ABB RAPID module: Module1.mod

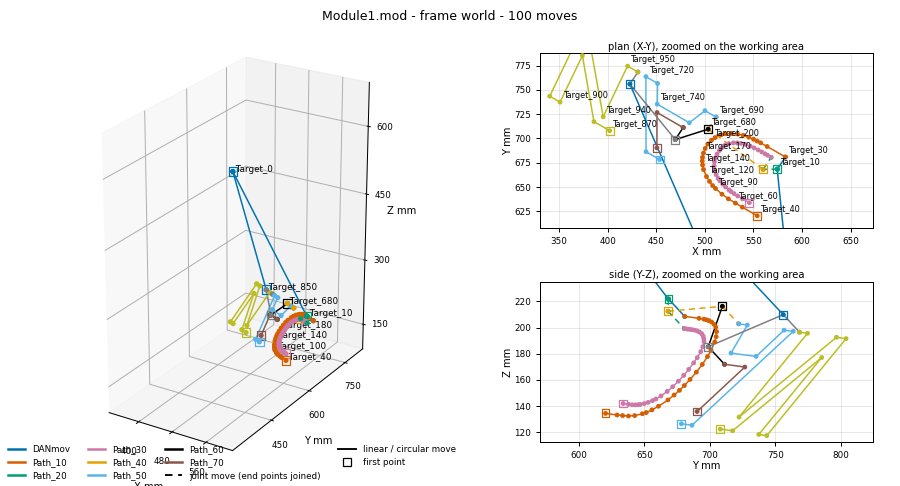
[picture p0: tool path of Module1.mod in frame world, 100 of 100 moves have a stored position in this frame; points joined in program order, loops and branches not executed]
MODULE Module1
        CONST robtarget Target_20:=[[0.071,0.06,-20],[1,0,0,0],[0,0,0,0],[9E+09,9E+09,9E+09,9E+09,9E+09,9E+09]];
    CONST robtarget Target_30:=[[0.095,0.07,0],[1,0,0,0],[0,0,0,0],[9E+09,9E+09,9E+09,9E+09,9E+09,9E+09]];
    CONST robtarget Target_40:=[[99.94,0.237,0],[1,0,0,0],[0,0,0,0],[9E+09,9E+09,9E+09,9E+09,9E+09,9E+09]];
    CONST robtarget Target_50:=[[99.89,17.95,0],[1,0,0,0],[0,0,0,0],[9E+09,9E+09,9E+09,9E+09,9E+09,9E+09]];
    CONST robtarget Target_60:=[[99.72,26.211,0],[1,0,0,0],[0,0,0,0],[9E+09,9E+09,9E+09,9E+09,9E+09,9E+09]];
    CONST robtarget Target_70:=[[99.369,34.775,0],[1,0,0,0],[0,0,0,0],[9E+09,9E+09,9E+09,9E+09,9E+09,9E+09]];
    CONST robtarget Target_80:=[[98.151,42.817,0],[1,0,0,0],[0,0,0,0],[9E+09,9E+09,9E+09,9E+09,9E+09,9E+09]];
    CONST robtarget Target_90:=[[95.465,51.41,0],[1,0,0,0],[0,0,0,0],[9E+09,9E+09,9E+09,9E+09,9E+09,9E+09]];
    CONST robtarget Target_100:=[[93.827,55.395,0],[1,0,0,0],[0,0,0,0],[9E+09,9E+09,9E+09,9E+09,9E+09,9E+09]];
    CONST robtarget Target_110:=[[90.626,60.139,0],[1,0,0,0],[0,0,0,0],[9E+09,9E+09,9E+09,9E+09,9E+09,9E+09]];
    CONST robtarget Target_120:=[[86.457,65.135,0],[1,0,0,0],[0,0,0,0],[9E+09,9E+09,9E+09,9E+09,9E+09,9E+09]];
    CONST robtarget Target_130:=[[79.404,71.019,0],[1,0,0,0],[0,0,0,0],[9E+09,9E+09,9E+09,9E+09,9E+09,9E+09]];
    CONST robtarget Target_140:=[[74.069,73.954,0],[1,0,0,0],[0,0,0,0],[9E+09,9E+09,9E+09,9E+09,9E+09,9E+09]];
    CONST robtarget Target_150:=[[69.003,75.99,0],[1,0,0,0],[0,0,0,0],[9E+09,9E+09,9E+09,9E+09,9E+09,9E+09]];
    CONST robtarget Target_160:=[[63.952,77.379,0],[1,0,0,0],[0,0,0,0],[9E+09,9E+09,9E+09,9E+09,9E+09,9E+09]];
    CONST robtarget Target_170:=[[57.546,78.369,0],[1,0,0,0],[0,0,0,0],[9E+09,9E+09,9E+09,9E+09,9E+09,9E+09]];
    CONST robtarget Target_180:=[[50.002,78.831,0],[1,0,0,0],[0,0,0,0],[9E+09,9E+09,9E+09,9E+09,9E+09,9E+09]];
    CONST robtarget Target_190:=[[42.114,78.338,0],[1,0,0,0],[0,0,0,0],[9E+09,9E+09,9E+09,9E+09,9E+09,9E+09]];
    CONST robtarget Target_200:=[[34.188,76.601,0],[1,0,0,0],[0,0,0,0],[9E+09,9E+09,9E+09,9E+09,9E+09,9E+09]];
    CONST robtarget Target_210:=[[27.953,74.421,0],[1,0,0,0],[0,0,0,0],[9E+09,9E+09,9E+09,9E+09,9E+09,9E+09]];
    CONST robtarget Target_220:=[[19.688,70.032,0],[1,0,0,0],[0,0,0,0],[9E+09,9E+09,9E+09,9E+09,9E+09,9E+09]];
    CONST robtarget Target_230:=[[14.672,66.13,0],[1,0,0,0],[0,0,0,0],[9E+09,9E+09,9E+09,9E+09,9E+09,9E+09]];
    CONST robtarget Target_240:=[[9.923,60.959,0],[1,0,0,0],[0,0,0,0],[9E+09,9E+09,9E+09,9E+09,9E+09,9E+09]];
    CONST robtarget Target_250:=[[5.883,54.79,0],[1,0,0,0],[0,0,0,0],[9E+09,9E+09,9E+09,9E+09,9E+09,9E+09]];
    CONST robtarget Target_260:=[[3.458,49.141,0],[1,0,0,0],[0,0,0,0],[9E+09,9E+09,9E+09,9E+09,9E+09,9E+09]];
    CONST robtarget Target_270:=[[1.636,43.084,0],[1,0,0,0],[0,0,0,0],[9E+09,9E+09,9E+09,9E+09,9E+09,9E+09]];
    CONST robtarget Target_280:=[[0.741,37.699,0],[1,0,0,0],[0,0,0,0],[9E+09,9E+09,9E+09,9E+09,9E+09,9E+09]];
    CONST robtarget Target_290:=[[0.334,33.582,0],[1,0,0,0],[0,0,0,0],[9E+09,9E+09,9E+09,9E+09,9E+09,9E+09]];
    CONST robtarget Target_300:=[[0.083,29.539,0],[1,0,0,0],[0,0,0,0],[9E+09,9E+09,9E+09,9E+09,9E+09,9E+09]];
    CONST robtarget Target_310:=[[-0.058,21.739,0],[1,0,0,0],[0,0,0,0],[9E+09,9E+09,9E+09,9E+09,9E+09,9E+09]];
    CONST robtarget Target_320:=[[-0.012,0.002,0],[1,0,0,0],[0,0,0,0],[9E+09,9E+09,9E+09,9E+09,9E+09,9E+09]];
    CONST robtarget Target_330:=[[0.01,0.019,-20],[1,0,0,0],[0,0,0,0],[9E+09,9E+09,9E+09,9E+09,9E+09,9E+09]];
    CONST robtarget Target_340:=[[11.428,13.269,-20],[1,0,0,0],[0,0,0,0],[9E+09,9E+09,9E+09,9E+09,9E+09,9E+09]];
    CONST robtarget Target_350:=[[11.415,13.206,0],[1,0,0,0],[0,0,0,0],[9E+09,9E+09,9E+09,9E+09,9E+09,9E+09]];
    CONST robtarget Target_360:=[[88.506,13.381,0],[1,0,0,0],[0,0,0,0],[9E+09,9E+09,9E+09,9E+09,9E+09,9E+09]];
    CONST robtarget Target_370:=[[88.487,21.649,0],[1,0,0,0],[0,0,0,0],[9E+09,9E+09,9E+09,9E+09,9E+09,9E+09]];
    CONST robtarget Target_380:=[[88.485,27.345,0],[1,0,0,0],[0,0,0,0],[9E+09,9E+09,9E+09,9E+09,9E+09,9E+09]];
    CONST robtarget Target_390:=[[88.109,31.752,0],[1,0,0,0],[0,0,0,0],[9E+09,9E+09,9E+09,9E+09,9E+09,9E+09]];
    CONST robtarget Target_400:=[[87.669,35.444,0],[1,0,0,0],[0,0,0,0],[9E+09,9E+09,9E+09,9E+09,9E+09,9E+09]];
    CONST robtarget Target_410:=[[87.109,38.017,0],[1,0,0,0],[0,0,0,0],[9E+09,9E+09,9E+09,9E+09,9E+09,9E+09]];
    CONST robtarget Target_420:=[[85.774,42.593,0],[1,0,0,0],[0,0,0,0],[9E+09,9E+09,9E+09,9E+09,9E+09,9E+09]];
    CONST robtarget Target_430:=[[84.168,46.535,0],[1,0,0,0],[0,0,0,0],[9E+09,9E+09,9E+09,9E+09,9E+09,9E+09]];
    CONST robtarget Target_440:=[[81.999,50.598,0],[1,0,0,0],[0,0,0,0],[9E+09,9E+09,9E+09,9E+09,9E+09,9E+09]];
    CONST robtarget Target_450:=[[80.078,53.34,0],[1,0,0,0],[0,0,0,0],[9E+09,9E+09,9E+09,9E+09,9E+09,9E+09]];
    CONST robtarget Target_460:=[[76.624,56.897,0],[1,0,0,0],[0,0,0,0],[9E+09,9E+09,9E+09,9E+09,9E+09,9E+09]];
    CONST robtarget Target_470:=[[71.616,60.336,0],[1,0,0,0],[0,0,0,0],[9E+09,9E+09,9E+09,9E+09,9E+09,9E+09]];
    CONST robtarget Target_480:=[[66.489,62.685,0],[1,0,0,0],[0,0,0,0],[9E+09,9E+09,9E+09,9E+09,9E+09,9E+09]];
    CONST robtarget Target_490:=[[60.688,64.314,0],[1,0,0,0],[0,0,0,0],[9E+09,9E+09,9E+09,9E+09,9E+09,9E+09]];
    CONST robtarget Target_500:=[[54.646,65.083,0],[1,0,0,0],[0,0,0,0],[9E+09,9E+09,9E+09,9E+09,9E+09,9E+09]];
    CONST robtarget Target_510:=[[48.445,65.222,0],[1,0,0,0],[0,0,0,0],[9E+09,9E+09,9E+09,9E+09,9E+09,9E+09]];
    CONST robtarget Target_520:=[[41.793,64.617,0],[1,0,0,0],[0,0,0,0],[9E+09,9E+09,9E+09,9E+09,9E+09,9E+09]];
    CONST robtarget Target_530:=[[36.504,63.714,0],[1,0,0,0],[0,0,0,0],[9E+09,9E+09,9E+09,9E+09,9E+09,9E+09]];
    CONST robtarget Target_540:=[[30.458,61.691,0],[1,0,0,0],[0,0,0,0],[9E+09,9E+09,9E+09,9E+09,9E+09,9E+09]];
    CONST robtarget Target_550:=[[25.646,58.958,0],[1,0,0,0],[0,0,0,0],[9E+09,9E+09,9E+09,9E+09,9E+09,9E+09]];
    CONST robtarget Target_560:=[[20.836,54.923,0],[1,0,0,0],[0,0,0,0],[9E+09,9E+09,9E+09,9E+09,9E+09,9E+09]];
    CONST robtarget Target_570:=[[18.13,51.34,0],[1,0,0,0],[0,0,0,0],[9E+09,9E+09,9E+09,9E+09,9E+09,9E+09]];
    CONST robtarget Target_580:=[[15.883,47.659,0],[1,0,0,0],[0,0,0,0],[9E+09,9E+09,9E+09,9E+09,9E+09,9E+09]];
    CONST robtarget Target_590:=[[13.855,43.017,0],[1,0,0,0],[0,0,0,0],[9E+09,9E+09,9E+09,9E+09,9E+09,9E+09]];
    CONST robtarget Target_600:=[[12.476,37.696,0],[1,0,0,0],[0,0,0,0],[9E+09,9E+09,9E+09,9E+09,9E+09,9E+09]];
    CONST robtarget Target_610:=[[11.809,33.29,0],[1,0,0,0],[0,0,0,0],[9E+09,9E+09,9E+09,9E+09,9E+09,9E+09]];
    CONST robtarget Target_620:=[[11.395,28.602,0],[1,0,0,0],[0,0,0,0],[9E+09,9E+09,9E+09,9E+09,9E+09,9E+09]];
    CONST robtarget Target_630:=[[11.309,24.432,0],[1,0,0,0],[0,0,0,0],[9E+09,9E+09,9E+09,9E+09,9E+09,9E+09]];
    CONST robtarget Target_640:=[[11.306,20.553,0],[1,0,0,0],[0,0,0,0],[9E+09,9E+09,9E+09,9E+09,9E+09,9E+09]];
    CONST robtarget Target_650:=[[11.368,17.578,0],[1,0,0,0],[0,0,0,0],[9E+09,9E+09,9E+09,9E+09,9E+09,9E+09]];
    CONST robtarget Target_660:=[[11.3,13.377,0],[1,0,0,0],[0,0,0,0],[9E+09,9E+09,9E+09,9E+09,9E+09,9E+09]];
    CONST robtarget Target_670:=[[11.431,13.345,-20],[1,0,0,0],[0,0,0,0],[9E+09,9E+09,9E+09,9E+09,9E+09,9E+09]];
    CONST robtarget Target_680:=[[-0.137,82.54,-20],[1,0,0,0],[0,0,0,0],[9E+09,9E+09,9E+09,9E+09,9E+09,9E+09]];
    CONST robtarget Target_690:=[[-0.154,82.529,0],[1,0,0,0],[0,0,0,0],[9E+09,9E+09,9E+09,9E+09,9E+09,9E+09]];
    CONST robtarget Target_700:=[[99.658,116.481,0],[1,0,0,0],[0,0,0,0],[9E+09,9E+09,9E+09,9E+09,9E+09,9E+09]];
    CONST robtarget Target_710:=[[99.61,132.697,0],[1,0,0,0],[0,0,0,0],[9E+09,9E+09,9E+09,9E+09,9E+09,9E+09]];
    CONST robtarget Target_720:=[[-0.345,166.23,0],[1,0,0,0],[0,0,0,0],[9E+09,9E+09,9E+09,9E+09,9E+09,9E+09]];
    CONST robtarget Target_730:=[[-0.179,152.289,0],[1,0,0,0],[0,0,0,0],[9E+09,9E+09,9E+09,9E+09,9E+09,9E+09]];
    CONST robtarget Target_740:=[[27.683,143.366,0],[1,0,0,0],[0,0,0,0],[9E+09,9E+09,9E+09,9E+09,9E+09,9E+09]];
    CONST robtarget Target_750:=[[27.893,105.098,0],[1,0,0,0],[0,0,0,0],[9E+09,9E+09,9E+09,9E+09,9E+09,9E+09]];
    CONST robtarget Target_760:=[[-0.159,95.872,0],[1,0,0,0],[0,0,0,0],[9E+09,9E+09,9E+09,9E+09,9E+09,9E+09]];
    CONST robtarget Target_770:=[[-0.14,82.55,0],[1,0,0,0],[0,0,0,0],[9E+09,9E+09,9E+09,9E+09,9E+09,9E+09]];
    CONST robtarget Target_780:=[[-0.154,82.561,-20],[1,0,0,0],[0,0,0,0],[9E+09,9E+09,9E+09,9E+09,9E+09,9E+09]];
    CONST robtarget Target_790:=[[39.082,108.722,-20],[1,0,0,0],[0,0,0,0],[9E+09,9E+09,9E+09,9E+09,9E+09,9E+09]];
    CONST robtarget Target_800:=[[39.077,108.691,0],[1,0,0,0],[0,0,0,0],[9E+09,9E+09,9E+09,9E+09,9E+09,9E+09]];
    CONST robtarget Target_810:=[[86.241,124.237,0],[1,0,0,0],[0,0,0,0],[9E+09,9E+09,9E+09,9E+09,9E+09,9E+09]];
    CONST robtarget Target_820:=[[38.992,139.852,0],[1,0,0,0],[0,0,0,0],[9E+09,9E+09,9E+09,9E+09,9E+09,9E+09]];
    CONST robtarget Target_830:=[[39.046,108.686,0],[1,0,0,0],[0,0,0,0],[9E+09,9E+09,9E+09,9E+09,9E+09,9E+09]];
    CONST robtarget Target_840:=[[39.049,108.56,-20],[1,0,0,0],[0,0,0,0],[9E+09,9E+09,9E+09,9E+09,9E+09,9E+09]];
    CONST robtarget Target_850:=[[-0.358,175.771,-20],[1,0,0,0],[0,0,0,0],[9E+09,9E+09,9E+09,9E+09,9E+09,9E+09]];
    CONST robtarget Target_860:=[[-0.349,175.774,0],[1,0,0,0],[0,0,0,0],[9E+09,9E+09,9E+09,9E+09,9E+09,9E+09]];
    CONST robtarget Target_870:=[[99.545,176.056,0],[1,0,0,0],[0,0,0,0],[9E+09,9E+09,9E+09,9E+09,9E+09,9E+09]];
    CONST robtarget Target_880:=[[99.462,194.82,0],[1,0,0,0],[0,0,0,0],[9E+09,9E+09,9E+09,9E+09,9E+09,9E+09]];
    CONST robtarget Target_890:=[[20.206,234.954,0],[1,0,0,0],[0,0,0,0],[9E+09,9E+09,9E+09,9E+09,9E+09,9E+09]];
    CONST robtarget Target_900:=[[99.467,235.15,0],[1,0,0,0],[0,0,0,0],[9E+09,9E+09,9E+09,9E+09,9E+09,9E+09]];
    CONST robtarget Target_910:=[[99.468,247.445,0],[1,0,0,0],[0,0,0,0],[9E+09,9E+09,9E+09,9E+09,9E+09,9E+09]];
    CONST robtarget Target_920:=[[-0.422,247.2,0],[1,0,0,0],[0,0,0,0],[9E+09,9E+09,9E+09,9E+09,9E+09,9E+09]];
    CONST robtarget Target_930:=[[-0.414,232.573,0],[1,0,0,0],[0,0,0,0],[9E+09,9E+09,9E+09,9E+09,9E+09,9E+09]];
    CONST robtarget Target_940:=[[85.947,188.296,0],[1,0,0,0],[0,0,0,0],[9E+09,9E+09,9E+09,9E+09,9E+09,9E+09]];
    CONST robtarget Target_950:=[[-0.342,188.055,0],[1,0,0,0],[0,0,0,0],[9E+09,9E+09,9E+09,9E+09,9E+09,9E+09]];
    CONST robtarget Target_960:=[[-0.342,175.796,0],[1,0,0,0],[0,0,0,0],[9E+09,9E+09,9E+09,9E+09,9E+09,9E+09]];
    CONST robtarget Target_970:=[[-0.334,175.799,-20],[1,0,0,0],[0,0,0,0],[9E+09,9E+09,9E+09,9E+09,9E+09,9E+09]];
    CONST robtarget Target_0:=[[-134.031,-231.216,-517.135],[1,0,0,0],[0,0,-1,0],[9E+09,9E+09,9E+09,9E+09,9E+09,9E+09]];
    CONST robtarget Target_10:=[[0.269,0.222,-20],[1,0,0,0],[0,0,0,0],[9E+09,9E+09,9E+09,9E+09,9E+09,9E+09]];
    CONST robtarget Target_1000:=[[-134.031,-231.216,-517.135],[1,0,0,0],[0,0,-1,0],[9E+09,9E+09,9E+09,9E+09,9E+09,9E+09]];
        TASK PERS wobjdata DANinclindo:=[FALSE,TRUE,"",[[0,0,10],[1,0,0,0]],[[366.1,610.764,198.883],[0.288677,-0.643742,0.654749,0.271228]]];
!***********************************************************
    !
    ! Módulo:  Module1
    !
    ! Descripción:
    !   <Introduzca la descripción aquí>
    !
    ! Autor: Danilo
    !
    ! Versión: 1.0
    !
    !***********************************************************


    !***********************************************************
    !
    ! Procedimiento Main
    !
    !   Este es el punto de entrada de su programa
    !
    !***********************************************************
    PROC main()
        !Añada aquí su código
        DANmov;
        Path_10;
        Path_20;
        Path_30;
        Path_40;
        Path_50;
        Path_60;
        Path_70;
        Path_80;
        Path_90;
        Path_100;
    ENDPROC
    PROC DANmov()
        MoveL Target_0,v100,z10,MARCADORBIEN\WObj:=DAN;
        MoveL Target_10,v100,z10,MARCADORBIEN\WObj:=DAN;
        MoveL Target_20,v100,z10,MARCADORBIEN\WObj:=DAN;
        MoveL Target_30,v100,z10,MARCADORBIEN\WObj:=DAN;
    ENDPROC
    PROC Path_10()
        MoveL Target_40,v100,z10,MARCADORBIEN\WObj:=DAN;
        MoveL Target_50,v100,z10,MARCADORBIEN\WObj:=DAN;
        MoveL Target_60,v100,z10,MARCADORBIEN\WObj:=DAN;
        MoveL Target_70,v100,z10,MARCADORBIEN\WObj:=DAN;
        MoveL Target_80,v100,z10,MARCADORBIEN\WObj:=DAN;
        MoveL Target_90,v100,z10,MARCADORBIEN\WObj:=DAN;
        MoveL Target_100,v100,z10,MARCADORBIEN\WObj:=DAN;
        MoveL Target_110,v100,z10,MARCADORBIEN\WObj:=DAN;
        MoveL Target_120,v100,z10,MARCADORBIEN\WObj:=DAN;
        MoveL Target_130,v100,z10,MARCADORBIEN\WObj:=DAN;
        MoveL Target_140,v100,z10,MARCADORBIEN\WObj:=DAN;
        MoveL Target_150,v100,z10,MARCADORBIEN\WObj:=DAN;
        MoveL Target_160,v100,z10,MARCADORBIEN\WObj:=DAN;
        MoveL Target_170,v100,z10,MARCADORBIEN\WObj:=DAN;
        MoveL Target_180,v100,z10,MARCADORBIEN\WObj:=DAN;
        MoveL Target_190,v100,z10,MARCADORBIEN\WObj:=DAN;
        MoveL Target_200,v100,z10,MARCADORBIEN\WObj:=DAN;
        MoveL Target_210,v100,z10,MARCADORBIEN\WObj:=DAN;
        MoveL Target_220,v100,z10,MARCADORBIEN\WObj:=DAN;
        MoveL Target_230,v100,z10,MARCADORBIEN\WObj:=DAN;
        MoveL Target_240,v100,z10,MARCADORBIEN\WObj:=DAN;
        MoveL Target_250,v100,z10,MARCADORBIEN\WObj:=DAN;
        MoveL Target_260,v100,z10,MARCADORBIEN\WObj:=DAN;
        MoveL Target_270,v100,z10,MARCADORBIEN\WObj:=DAN;
        MoveL Target_280,v100,z10,MARCADORBIEN\WObj:=DAN;
        MoveL Target_290,v100,z10,MARCADORBIEN\WObj:=DAN;
        MoveL Target_300,v100,z10,MARCADORBIEN\WObj:=DAN;
        MoveL Target_310,v100,z10,MARCADORBIEN\WObj:=DAN;
        MoveL Target_320,v100,z10,MARCADORBIEN\WObj:=DAN;
    ENDPROC
    PROC Path_20()
        MoveJ Target_330,v100,z10,MARCADORBIEN\WObj:=DAN;
        MoveJ Target_340,v100,z10,MARCADORBIEN\WObj:=DAN;
        MoveJ Target_350,v100,z10,MARCADORBIEN\WObj:=DAN;
    ENDPROC
    PROC Path_30()
        MoveL Target_360,v100,z10,MARCADORBIEN\WObj:=DAN;
        MoveL Target_370,v100,z10,MARCADORBIEN\WObj:=DAN;
        MoveL Target_380,v100,z10,MARCADORBIEN\WObj:=DAN;
        MoveL Target_390,v100,z10,MARCADORBIEN\WObj:=DAN;
        MoveL Target_400,v100,z10,MARCADORBIEN\WObj:=DAN;
        MoveL Target_410,v100,z10,MARCADORBIEN\WObj:=DAN;
        MoveL Target_420,v100,z10,MARCADORBIEN\WObj:=DAN;
        MoveL Target_430,v100,z10,MARCADORBIEN\WObj:=DAN;
        MoveL Target_440,v100,z10,MARCADORBIEN\WObj:=DAN;
        MoveL Target_450,v100,z10,MARCADORBIEN\WObj:=DAN;
        MoveL Target_460,v100,z10,MARCADORBIEN\WObj:=DAN;
        MoveL Target_470,v100,z10,MARCADORBIEN\WObj:=DAN;
        MoveL Target_480,v100,z10,MARCADORBIEN\WObj:=DAN;
        MoveL Target_490,v100,z10,MARCADORBIEN\WObj:=DAN;
        MoveL Target_500,v100,z10,MARCADORBIEN\WObj:=DAN;
        MoveL Target_510,v100,z10,MARCADORBIEN\WObj:=DAN;
        MoveL Target_520,v100,z10,MARCADORBIEN\WObj:=DAN;
        MoveL Target_530,v100,z10,MARCADORBIEN\WObj:=DAN;
        MoveL Target_540,v100,z10,MARCADORBIEN\WObj:=DAN;
        MoveL Target_550,v100,z10,MARCADORBIEN\WObj:=DAN;
        MoveL Target_560,v100,z10,MARCADORBIEN\WObj:=DAN;
        MoveL Target_570,v100,z10,MARCADORBIEN\WObj:=DAN;
        MoveL Target_580,v100,z10,MARCADORBIEN\WObj:=DAN;
        MoveL Target_590,v100,z10,MARCADORBIEN\WObj:=DAN;
        MoveL Target_600,v100,z10,MARCADORBIEN\WObj:=DAN;
        MoveL Target_610,v100,z10,MARCADORBIEN\WObj:=DAN;
        MoveL Target_620,v100,z10,MARCADORBIEN\WObj:=DAN;
        MoveL Target_630,v100,z10,MARCADORBIEN\WObj:=DAN;
        MoveL Target_640,v100,z10,MARCADORBIEN\WObj:=DAN;
        MoveL Target_650,v100,z10,MARCADORBIEN\WObj:=DAN;
        MoveL Target_660,v100,z10,MARCADORBIEN\WObj:=DAN;
    ENDPROC
    PROC Path_40()
        MoveJ Target_670,v50,z10,MARCADORBIEN\WObj:=DAN;
        MoveJ Target_680,v50,z10,MARCADORBIEN\WObj:=DAN;
        MoveJ Target_680,v50,z10,MARCADORBIEN\WObj:=DAN;
        MoveJ Target_690,v50,z10,MARCADORBIEN\WObj:=DAN;
    ENDPROC
    PROC Path_50()
        MoveL Target_700,v100,z10,MARCADORBIEN\WObj:=DAN;
        MoveL Target_710,v100,z10,MARCADORBIEN\WObj:=DAN;
        MoveL Target_720,v100,z10,MARCADORBIEN\WObj:=DAN;
        MoveL Target_730,v100,z10,MARCADORBIEN\WObj:=DAN;
        MoveL Target_740,v100,z10,MARCADORBIEN\WObj:=DAN;
        MoveL Target_750,v100,z10,MARCADORBIEN\WObj:=DAN;
        MoveL Target_760,v100,z10,MARCADORBIEN\WObj:=DAN;
        MoveL Target_770,v100,z10,MARCADORBIEN\WObj:=DAN;
    ENDPROC
    PROC Path_60()
        MoveL Target_780,v50,z10,MARCADORBIEN\WObj:=DAN;
        MoveL Target_790,v50,z10,MARCADORBIEN\WObj:=DAN;
        MoveL Target_800,v50,z10,MARCADORBIEN\WObj:=DAN;
    ENDPROC
    PROC Path_70()
        MoveL Target_810,v100,z10,MARCADORBIEN\WObj:=DAN;
        MoveL Target_820,v100,z10,MARCADORBIEN\WObj:=DAN;
        MoveL Target_830,v100,z10,MARCADORBIEN\WObj:=DAN;
    ENDPROC
    PROC Path_80()
        MoveL Target_840,v50,z10,MARCADORBIEN\WObj:=DAN;
        MoveL Target_850,v50,z10,MARCADORBIEN\WObj:=DAN;
        MoveL Target_860,v50,z10,MARCADORBIEN\WObj:=DAN;
    ENDPROC
    PROC Path_90()
        MoveL Target_870,v100,z10,MARCADORBIEN\WObj:=DAN;
        MoveL Target_880,v100,z10,MARCADORBIEN\WObj:=DAN;
        MoveL Target_890,v100,z10,MARCADORBIEN\WObj:=DAN;
        MoveL Target_900,v100,z10,MARCADORBIEN\WObj:=DAN;
        MoveL Target_910,v100,z10,MARCADORBIEN\WObj:=DAN;
        MoveL Target_920,v100,z10,MARCADORBIEN\WObj:=DAN;
        MoveL Target_930,v100,z10,MARCADORBIEN\WObj:=DAN;
        MoveL Target_940,v100,z10,MARCADORBIEN\WObj:=DAN;
        MoveL Target_950,v100,z10,MARCADORBIEN\WObj:=DAN;
        MoveL Target_960,v100,z10,MARCADORBIEN\WObj:=DAN;
    ENDPROC
    PROC Path_100()
        MoveL Target_970,v100,z10,MARCADORBIEN\WObj:=DAN;
        MoveL Target_1000,v50,z10,MARCADORBIEN\WObj:=DAN;
    ENDPROC
ENDMODULE
